// TIA Portal V20 export
TYPE "UDT_RunTime_Status"
   STRUCT
      Run_Time : Struct
         Seconds : Int;
         Minutes : Int;
         Hours : Real;
         Days : Real;
         Years : Real;
      END_STRUCT;
   END_STRUCT;
END_TYPE
